17729	:	NCErrorSTRING :='"Axis address" Controller does not know its axis, or the axis address has not been initialized.	.';
17730	:	NCErrorSTRING :='"Drive address" Controller does not know its drive, or the drive address has not been initialized.	.';
17744	:	NCErrorSTRING :='"Following error monitoring (position)" With active following error monitoring (position) a following error exceedance has occurred, whose magnitude is greater than the following error window, and whose duration is longer than the parameterized following error filter time.	.';
17745	:	NCErrorSTRING :='"Following error monitoring (velocity)" With active following error monitoring (velocity) a velocity following error exceedance has occurred, whose magnitude is greater than the following error window, and whose duration is longer than the parameterized following error filter time.	.';
17824	:	NCErrorSTRING :='"CONTROLERR_RANGE_AREA_ASIDE"	.';
17825	:	NCErrorSTRING :='"CONTROLERR_RANGE_AREA_BSIDE"	.';
17826	:	NCErrorSTRING :='"CONTROLERR_RANGE_QNENN"	.';
17827	:	NCErrorSTRING :='"CONTROLERR_RANGE_PNENN"	.';
17828	:	NCErrorSTRING :='"CONTROLERR_RANGE_AXISIDPRESP0"	.';
17920	:	NCErrorSTRING :='‘"Drive ID not allowed" The value for the drive ID is not allowed, e.g. because it has already been assigned, is less than or equal to zero, or is greater than 255.	.';
17921	:	NCErrorSTRING :='‘Drive type impermissible’ The value for the drive type is impermissible, since it is not defined.	.';
17922	:	NCErrorSTRING :='‘Drive operating mode impermissible’ The value for the drive operating mode is impermissible (mode 1: standard).	.';
17923	:	NCErrorSTRING :='"Motor polarity inverted?" The flag for the motor polarity is not allowed. Flag 0: Positive motor polarity flag 1: Negative motor polarity	.';
17924	:	NCErrorSTRING :='‘Drift compensation/speed offset (DAC offset)’ The value for the drift compensation (DAC offset) is impermissible.	.';
17925	:	NCErrorSTRING :='‘Reference speed (velocity pre-control)’ The value for the reference speed (also called velocity pilot control) is impermissible.	.';
17926	:	NCErrorSTRING :='‘Reference output in percent’ The value for the reference output in percent is impermissible. The value 1.0 (100 %) usually corresponds to a voltage of 10.0 V.	.';
17927	:	NCErrorSTRING :='‘Quadrant compensation factor’ The value for the quadrant compensation factor is impermissible.	.';
17928	:	NCErrorSTRING :='‘Velocity reference point’ The value for the velocity reference point in percent is impermissible. The value 1.0 corresponds to 100 percent.	.';
17929	:	NCErrorSTRING :='‘Output reference point’ The value for the output reference point in percent is impermissible. The value 1.0 corresponds to 100 percent.	.';
17930	:	NCErrorSTRING :='‘Minimum or maximum output limits (output limitation)’ The value for the minimum and/or maximum output limit is impermissible. This will happen if the range of values is exceeded, the maximum limit is smaller than the minimum limit, or the distance between the minimum and maximum limits is zero.';
17931	:	NCErrorSTRING :='"Parameter “Maximum Value for Output” is Improper The value for the maximum number of output digits of motion controllers (maximum output value) is improper. According to the used interface (e.g. position, velocity or torque/current). Regarding a velocity interface it is often about a signed 16 bit output value (± 32767)."	.';
17932	:	NCErrorSTRING :='"Parameter “Internal Drive Control Word” is Improper The value as Internal Drive Control Word for the NC is improper. In this control word information from the system manager to the NC is contained what is evaluated at the TC start of the NC."	.';
17933	:	NCErrorSTRING :='"Parameter “Internal Timer for RESET Behavior of Motion Controller” is Improper The special parameter that influences the internal timing behavior between the NC motion controller and the IO motion controller is improper."	.';
17934	:	NCErrorSTRING :='"Parameter “Master Motion Controller ID” is Improper The parameter “master motion controller ID” is improper for a further NC motion controller in slave mode.';
17935	:	NCErrorSTRING :='‘Drive torque output scaling impermissible’ The value is impermissible as drive torque output scaling (rotary motor) or as force output scaling (linear motor).	.';
17936	:	NCErrorSTRING :='„Drive velocity output scaling is not allowed“ The value for the drive velocity output scaling is not allowed.	.';
17937	:	NCErrorSTRING :='‘Profi Drive DSC proportional gain Kpc (controller) impermissible’ Positions The value for the Profi Drive DSC position control gain (Kpc factor) is impermissible.	.';
17938	:	NCErrorSTRING :='‘Table ID is impermissible’ The value for the table ID is impermissible.	.';
17939	:	NCErrorSTRING :='‘Table interpolation type is impermissible’ The value is impermissible as the table interpolation type.	.';
17940	:	NCErrorSTRING :='‘Output offset in percent is impermissible’ The value is impermissible as an output offset in percent (+/- 1.0).	.';
17941	:	NCErrorSTRING :='"‘Profi Drive DSC scaling for calculation of “Xerr” (controller) impermissible’ Positions: the value is impermissible as Profi Drive DSC scaling for the calculation of ‘Xerr’."	.';
17942	:	NCErrorSTRING :='‘Drive acceleration output scaling impermissible’ The value is impermissible as drive acceleration/deceleration output scaling.	.';
17943	:	NCErrorSTRING :='‘Drive position output scaling impermissible’ The value is impermissible as drive position output scaling.	.';
17944	:	NCErrorSTRING :='"Parameter “Dead Time Compensation Mode” (Motion Controller) is Invalid The parameter for the mode of dead time compensation of NC motion controllers is invalid (OFF, ON with velocity, ON with velocity and acceleration)."	.';
17945	:	NCErrorSTRING :='"Parameter “Control Bits of Dead Time Compensation” (Motion Controller) is Invalid The parameter for “control bits of dead time compensation” of NC motion controllers is invalid (e.g. relative or absolute time interpretation)."	.';
17946	:	NCErrorSTRING :='"Parameter “Time Shift of Dead Time Compensation” (Motion Controller) is Invalid The parameter for the time shift of dead time compensation (time shift in nanoseconds) of the NC motion controller is invalid."	.';
17947	:	NCErrorSTRING :='"Parameter “Output Delay (Velocity)” is Invalid The parameter for an optional output delay within the velocity interface to the motion controller is invalid (output delay (velocity)). The maximum permitted delay time has to be smaller than 100 times the NC SAF cycle time."	.';
17948	:	NCErrorSTRING :='‘Drive filter type impermissible for command variable filter for the output position’ The value is impermissible as a drive filter type for the smoothing of the output position (command variable filter for the setpoint position).	.';
17949	:	NCErrorSTRING :='‘Drive filter time impermissible for command variable filter for the output position’ The value is impermissible as a drive filter time for the smoothing of the output position (command variable filter for the setpoint position).	.';
17950	:	NCErrorSTRING :='‘Drive filter order impermissible for command variable filter for the output position’ The value is impermissible as a drive filter order (P-Tn) for the smoothing of the output position (command variable filter for the setpoint position).	.';
17952	:	NCErrorSTRING :='‘Bit mask for stepper motor cycle impermissible’ A value of the different stepper motor masks is impermissible for the respective cycle.	.';
17953	:	NCErrorSTRING :='‘Bit mask for stepper motor holding current impermissible’ The value for the stepper motor holding mask is impermissible.	.';
17954	:	NCErrorSTRING :='‘Scaling factor for actual torque (actual current) impermissible’ The value is impermissible as a scaling factor for the actual torque (or actual current).	.';
17955	:	NCErrorSTRING :='‘Filter time for actual torque is impermissible’ The value is impermissible as a filter time for the actual torque (or the actual current) (P-T1 filter).	.';
17956	:	NCErrorSTRING :='‘Filter time for the temporal derivation of the actual torque is impermissible’ The value is impermissible as a filter time for the temporal derivation of the actual torque (or actual current (P-T1 filter).	.';
17957	:	NCErrorSTRING :='"Parameter for the “Motion Controller Operation Mode” is Invalid The parameter for the motion controller operation mode (position mode, velocity mode, torque mode, …) is invalid.';
17958	:	NCErrorSTRING :='"Motion Controller Functionality is Not Supported A motion controller functionality has been set off that has not been released for usage or has not been implemented (e.g. writing or reading of a motion controller mode that is not supported by certain motion controllers).';
17959	:	NCErrorSTRING :='DRIVEOPERATIONMODEBUSY. The activation of the motion controller controlling mode has failed because another object with OID… uses this interface already.	.';
17960	:	NCErrorSTRING :='"Motion Controller Operation Mode Switching has not been configured or the desired motion controller operation mode cannot be found There has not any motion controller operation mode switching been configured and thus no reading or writing of a motion controller operation mode is possible.';
17968	:	NCErrorSTRING :='‘Overtemperature’ Overtemperature was detected or reported in the drive or terminal.	.';
17969	:	NCErrorSTRING :='‘Undervoltage’ Undervoltage was detected or reported in the drive or terminal.	.';
17970	:	NCErrorSTRING :='‘Wire break in phase A’ A wire break in phase A was detected or reported in the drive or terminal.	.';
17971	:	NCErrorSTRING :='‘Wire break in phase B’ A wire break in phase B was detected or reported in the drive or terminal.	.';
17972	:	NCErrorSTRING :='‘Overcurrent in phase A’ Overcurrent was detected or reported in phase A in the drive or terminal.	.';
17973	:	NCErrorSTRING :='‘Overcurrent in phase B’ Overcurrent was detected or reported in phase B in the drive or terminal.	.';
17974	:	NCErrorSTRING :='‘Torque overload (stall)’ A torque overload (stall) was detected or reported in the drive or terminal.	.';
17984	:	NCErrorSTRING :='‘Drive initialization’ Drive has not been initialized.  Although the drive has been created, the rest of the initialization has not been performed (1. Initialization of drive I/O, 2. Initialization of drive, 3. Reset drive).	.';
17985	:	NCErrorSTRING :='‘Axis address’ Drive does not know its axis, or the axis address has not been initialized.	.';
17986	:	NCErrorSTRING :='‘Address IO input structure’ Drive has no valid IO input address in the process image.	.';
17987	:	NCErrorSTRING :='‘Address IO output structure’ Drive has no valid IO output address in the process image.	.';
18000	:	NCErrorSTRING :='Drive hardware not ready to operate - the drive is in the error state (hardware error)';
18001	:	NCErrorSTRING :='Error in the cyclic communication OF the drive (Life Counter). Reasons FOR THIS could be an interrupted fieldbus OR a drive that is in the error state.	.';
18002	:	NCErrorSTRING :='‘Changing the table ID when active controller enable is impermissible’. Changing (deselecting, selecting) the characteristic curve table ID is not permissible when the controller enable for the axis is active.	.';
18005	:	NCErrorSTRING :='"‘Invalid IO data for more than ‘n’ continuous NC cycles’ The axis (encoder or drive) has detected invalid IO data (e.g. n=3) for more than ‘n’ continuous NC cycles (NC SAF task).';
18944	:	NCErrorSTRING :='"Table ID not allowed" The value for the table ID is not allowed, e.g. because it has already been assigned, is less than or equal to zero, or is greater than 255.	.';
18945	:	NCErrorSTRING :='"Table type not allowed" The value for the table type is unacceptable because it is not defined.	.';
18946	:	NCErrorSTRING :='"Number of lines in the table not allowed" The value of the number of lines in the table is not allowed, because, for example, it is smaller than two at linear interpolation and smaller than four at spline interpolation.	.';
18947	:	NCErrorSTRING :='"Number of columns in the table is not allowed" The value of the number of columns in the table is not allowed, because, for example, it is less than or equal to zero (depends upon the type of table or slave).	.';
18948	:	NCErrorSTRING :='"Step size (position delta) not allowed" The value for the step size between two lines (position delta) is not allowed, because, for example, it is less than or equal to zero.	.';
18949	:	NCErrorSTRING :='"Period not allowed" The value for the period is not allowed, because, for example, it is less than or equal to zero.	.';
18950	:	NCErrorSTRING :='"Table is not monotonic" The value for the step size is not allowed, because, for example, it is less than or equal to zero.	.';
18951	:	NCErrorSTRING :='„Table sub type is not allowed“ The value for the table sub type is not allowed or otherwise the table class (slave type) do not match up to the table main type. Table sub type: (1) equidistant linear position table, (2) equidistant cyclic position table, (3) none equidistant linear position table, (4) none equidistant cyclic position table	.';
18952	:	NCErrorSTRING :='„Table interpolation type is not allowed“ The value for the table interpolation type is allowed. Table interpolation type: (0) linear-interpolation, (1) 4-point-interpolation, (2) spline-interpolation	.';
18953	:	NCErrorSTRING :='"Incorrect table main type" The table main type is unknown or otherwise the table class (slave type) do not match up to the table main type. Table main type: (1) camming table, (2) characteristic table, (3) motion function table (MF)	.';
18960	:	NCErrorSTRING :='"Table initialization" Table has not been initialized. Although the table has been created, the rest of the initialization has not been performed. For instance, the number of lines or columns may be less than or equal to zero.	.';
18961	:	NCErrorSTRING :='"Not enough memory" Table could not be created, since there is not enough memory.	.';
18962	:	NCErrorSTRING :='"Function not executed, function not available" The function has not been implemented, or cannot be executed, for the present type of table.	.';
18963	:	NCErrorSTRING :='"Line index not allowed" The start line index or the stop line index to be used for read or write access to the table is not allowed. For instance, the line index may be greater than the total number of lines in the table.	.';
18964	:	NCErrorSTRING :='"Column index not allowed" The start column index or the stop column index to be used for read or write access to the table in not allowed. For instance, the column index may be greater than the total number of columns in the table.	.';
18965	:	NCErrorSTRING :='"Number of lines not allowed" The number of lines to be read from or written to the table is not allowed. The number of lines must be an integer multiple of the number of elements in a line (n * number of columns).	.';
18966	:	NCErrorSTRING :='"Number of columns not allowed" The number of columns to be read from or written to the table is not allowed. The number of columns must be an integer multiple of the number of elements in a column (n * number of lines).	.';
18967	:	NCErrorSTRING :='"Error in scaling or in range entry" The entries in the table header are inconsistent, e.g. the validity range is empty. If the error is generated during the run time it is a run time error and stops the master/slave group.	.';
18968	:	NCErrorSTRING :='"Multi table slave out of range" The slave master position is outside the table values for the master. The error is a run- time error, and stops the master/slave group.	.';
18969	:	NCErrorSTRING :='"Solo table underflow" The slave master position is outside the table values for the master. The master value of the equidistant table, to be processed linearly, lies under the first table value. The error is a run-time error, and stops the master/slave group.	.';
18970	:	NCErrorSTRING :='"Solo table overflow" The slave master position is outside the table values for the master. The master value of the equidistant table, to be processed linearly, lies above the first table value. The error is a run-time error, and stops the master/slave group.	.';
18971	:	NCErrorSTRING :='"Incorrect execution mode" The cyclic execution mode can only be "true" or "false".	.';
18972	:	NCErrorSTRING :='"Impermissible parameter" The Fifo parameter is not allowed.	.';
18973	:	NCErrorSTRING :='"Fifo is empty" The Fifo of the external generator is empty. This can signify end of track or a run time error.	.';
18974	:	NCErrorSTRING :='"Fifo is full" The Fifo of the external generator is full. It is the user‘s task to continue to attempt to fill the Fifo with the rejected values.	.';
18975	:	NCErrorSTRING :='"„Point-Index of Motion Function invalid“ The point index of a Motion Function Point of a Function Table is invalid. First the point index has to be larger than zero and second it has to be numerical continuously for one column in the Motion Function Table';
18976	:	NCErrorSTRING :='„No diagonalization of matrix“ The spline can not be calculated. The master positions are not correct.	.';
18977	:	NCErrorSTRING :='„Number of spline points to less“ The number of points of a cubic spline has to be greater than two.	.';
18978	:	NCErrorSTRING :='„Fifo must not be overwritten“ Fifo must not be overwritten since then the active line would be overwritten. It is the task of the user to secure that the active line is not modified.	.';
18979	:	NCErrorSTRING :='„Insufficient number of Motion Function points“ The number of valid Motion Function points is less than two. Either the entire number of points is to low or the point type of many points is set to Ignore Point.	.';
19200	:	NCErrorSTRING :='"Axis was stopped" The axis was stopped during travel to the target position. The axis may have been stopped with a PLC command via ADS, a call via AXFNC, or by the System Manager.	.';
19201	:	NCErrorSTRING :='"Axis cannot be started"';
19202	:	NCErrorSTRING :='"Control mode not permitted" No target position control, and no position range control.	.';
19203	:	NCErrorSTRING :='"Axis is not moving" The position and velocity can only be restarted while the axis is physically in motion.	.';
19204	:	NCErrorSTRING :='"“Invalid Mode” Examples: Invalid Direction input to MC_MoveModulo. Inactive axis parameter position correction for MC_BacklashCompensation."	.';
19205	:	NCErrorSTRING :='"Command not permitted"" •  Continuous motion in an unspecified direction •  Read/Write parameters: type mismatch"	.';
19206	:	NCErrorSTRING :='"Parameter incorrect"" •  Incorrect override: > 100% or < 0% •  Incorrect gear ratio: RatioDenominator = 0".';
19207	:	NCErrorSTRING :='"Timeout axis function block"" After positioning, all ""MC_Move..."" blocks check whether positioning was completed successfully. In the simplest case, the ""AxisHasJob"" flag of the NC axis is checked, which initially signifies that positioning was logically completed. ';
19208	:	NCErrorSTRING :='"Axis is in protected mode" The axis is in protected mode ( e.g. coupled) and cannot be moved.	.';
19209	:	NCErrorSTRING :='"Axis is not ready" The axis is not ready and cannot be moved.	.';
19210	:	NCErrorSTRING :='"Error during referencing" Referencing (homing) of the axis could not be started or was not successful.	.';
19211	:	NCErrorSTRING :='"Incorrect definition of the trigger input" The definition of the trigger signal for block MC_TouchProbe is incorrect. The defined encoder-ID, the trigger signal or the trigger edge are invalid.	.';
19212	:	NCErrorSTRING :='"Position latch was disabled" The function block MC_TouchProbe has detected that a measuring probe cycle it had started was disabled. The reason may be an axis reset, for example.	.';
19213	:	NCErrorSTRING :='‘NC status feedback timeout’  A function was successfully sent from the PLC to the NC. An expected feedback in the axis status word has not arrived.	.';
19214	:	NCErrorSTRING :='"Additional product not installed" The function is available as an additional product but is not installed on the system.	.';
19215	:	NCErrorSTRING :='"No NC Cycle Counter Update" – The NcToPlc Interface or the NC Cycle Counter in the NcToPlc Interface was not updated.	.';
19216	:	NCErrorSTRING :='"M-function query missing" This error occurs if the M- function was confirmed, but the request bit was not set.	.';
19217	:	NCErrorSTRING :='"Zero offset index is outside the range" The index of the zero offset is invalid.	.';
19218	:	NCErrorSTRING :='"R-parameter index or size is invalid" This error occurs if the R-parameters are written or read but the index or size are outside the range.	.';
19219	:	NCErrorSTRING :='"Index for tool description is invalid"	.';
19220	:	NCErrorSTRING :='"Version of the cyclic channel interface does not match the requested function or the function block" This error occurs if an older TwinCAT version is used to call new functions of a later TcNci.lib version.	.';
19221	:	NCErrorSTRING :='"Channel is not ready for the requested function" The requested function cannot be executed, because the channel is in the wrong state. This error occurs during reverse travel, for example, if the axis was not stopped with ItpEStop first.	.';
19222	:	NCErrorSTRING :='"Requested function is not activated" The requested function requires explicit activation.	.';
19223	:	NCErrorSTRING :='"Axis is already in another group" The axis has already been added to another group.	.';
19224	:	NCErrorSTRING :='"Block search could not be executed successfully"" The block search has failed. ';
19225	:	NCErrorSTRING :='"Invalid block search parameter" This error occurs if the FB ItpBlocksearch is called with invalid parameters (e.g. E_ItpDryRunMode, E_ItpBlockSearchMode)	.';
19232	:	NCErrorSTRING :='"Cannot add all axes" This error occurs if an auxiliary axis is to be added to an interpolation group, but the function fails. It is likely that a preceding instruction of an auxiliary axis was skipped.	.';
19248	:	NCErrorSTRING :='"Pointer is invalid"" A pointer to a data structure is invalid, e.g. Null•  Data structure MC_CAM_REF was not initialized"	.';
19249	:	NCErrorSTRING :='"Memory size invalid"" The specification of the memory size (SIZE) for a data structure is invalid.';
19250	:	NCErrorSTRING :='"Cam table ID is invalid" The ID of a cam table is not between 1 and 255.	.';
19251	:	NCErrorSTRING :='"Point ID is invalid" The ID of a point (sampling point) of a motion function is less than 1.	.';
19252	:	NCErrorSTRING :='"Number of points is invalid" The number of points (sampling points) of a cam plate to be read or written is less than 1.	.';
19253	:	NCErrorSTRING :='"MC table type is invalid" The type of a cam plate does not match the definition MC_TableType.	.';
19254	:	NCErrorSTRING :='"Number of rows invalid" The number of rows (sampling points) of a cam table is less than 1.	.';
19255	:	NCErrorSTRING :='"Number of columns invalid"" The number of columns of a cam table is invalid.';
19256	:	NCErrorSTRING :='"Step size invalid". The increment for the interpolation is invalid, e.g. less than or equal to zero.	.';
19264	:	NCErrorSTRING :='"Terminal type not supported" The terminal used is not supported by this function block.	.';
19265	:	NCErrorSTRING :='"Register read/write error" This error implies a validity error.	.';
19266	:	NCErrorSTRING :='"Axis is enabled" The axis is enabled but should not be enabled for this process.	.';
19267	:	NCErrorSTRING :='"Incorrect size of the compensation table" The specified table size (in bytes) does not match the actual size	.';
19268	:	NCErrorSTRING :='The minimum/maximum position in the compensation table does not match the position in the table description (ST_CompensationDesc)	.';
19269	:	NCErrorSTRING :='"Not implemented" The requested function is not implemented in this combination	.';
19296	:	NCErrorSTRING :='"Motion command did not become active" A motion command has been started and has been buffered and confirmed by the NC. Nevertheless, the motion command did not become active (possibly due to a terminating condition or an internal NC error).	.';
19297	:	NCErrorSTRING :='"Motion command could not be monitored by the PLC" A motion command has been started and has been buffered and confirmed by the NC. The PLC has not been able to monitor the execution of this command and the execution status is unclear since the NC is already executing a more recent command.';
19298	:	NCErrorSTRING :='"Buffered command was terminated with an error" A buffered command was terminated with an error. The error number is not available, because a new command is already being executed.	.';
19299	:	NCErrorSTRING :='"Buffered command was completed without feedback" A buffered command was completed but there was no feedback to indicate success or failure.	.';
19300	:	NCErrorSTRING :='"BufferMode is not supported by the command" The BufferMode is not supported by this command.	.';
19301	:	NCErrorSTRING :='"Command number is zero" The command number for queued commands managed by the system unexpectedly has the value 0.	.';
19302	:	NCErrorSTRING :='"Function block was not called cyclically" The function block was not called cyclically. The command execution could not be monitored by the PLC, because the NC was already executing a subsequent command. The execution state is unclear.	.';
19313	:	NCErrorSTRING :='"Invalid NCI entry type". The FB FB_NciFeedTablePreparation was called with an unknown nEntryType.	.';
19314	:	NCErrorSTRING :='"NCI feed table full"" The table is full, and the entry is therefore not accepted.';
19315	:	NCErrorSTRING :='INTERNAL error	.';
19316	:	NCErrorSTRING :='"ST_NciTangentialFollowingDesc: tangential axis is not an auxiliary axis" The entry for tangential following contains a tangential axis that is not an auxiliary axis.	.';
19317	:	NCErrorSTRING :='ST_NciTangentialFollowingDesc: nPathAxis1 or nPathAxis2 is not a path axis. It is therefore not possible to determine the plane.	.';
19318	:	NCErrorSTRING :='ST_NciTangentialFollwoingDesc: nPathAxis1 and nPathAxis2 are the same. It is therefore not possible to determine the plane.	.';
19319	:	NCErrorSTRING :='ST_NciGeoCirclePlane: Circle incorrectly parameterized	.';
19320	:	NCErrorSTRING :='Internal error during calculation of tangential following	.';
19321	:	NCErrorSTRING :='Tangential following: Monitoring of the deviation angle was activated during activation of tangential following (E_TfErrorOnCritical1), and an excessively large deviation angle was detected in the current segment.	.';
19322	:	NCErrorSTRING :='not implemented	.';
19323	:	NCErrorSTRING :='Tangential following: the radius of the current arc is too small	.';
19324	:	NCErrorSTRING :='FB_NciFeedTablePreparation: pEntry is NULL	.';
19325	:	NCErrorSTRING :='FB_NciFeedTablePreparation: the specified nEntryType does not match the structure type	.';
19326	:	NCErrorSTRING :='ST_NciMFuncFast and ST_NciMFuncHsk: the requested M-function is not between 0 and 159	.';
19327	:	NCErrorSTRING :='ST_NciDynOvr: the requested value for the dynamic override is not between 0.01 and 1	.';
19328	:	NCErrorSTRING :='ST_NciVertexSmoothing: invalid parameter. This error is generated if a negative smoothing radius or an unknown smoothing type is encountered.	.';
19329	:	NCErrorSTRING :='FB_NciFeedTablePrepartion: The requested velocity is not in the valid range	.';
19330	:	NCErrorSTRING :='ST_Nci*: invalid parameter	.';
19344	:	NCErrorSTRING :='Determined drive type is not supported	.';
19345	:	NCErrorSTRING :='Direction is impermissible	.';
19346	:	NCErrorSTRING :='SwitchMode is impermissible	.';
19347	:	NCErrorSTRING :='Mode for the parameter handling is impermissible	.';
19348	:	NCErrorSTRING :='Parameterization of the torque limits is inconsistent	.';
19349	:	NCErrorSTRING :='Parameterization of the position lag limit is impermissible (<=0).	.';
19350	:	NCErrorSTRING :='Parameterization of the distance limit is impermissible (<0)	.';
19351	:	NCErrorSTRING :='An attempt was made to back up parameters again, although they have already been backed up.	.';
19352	:	NCErrorSTRING :='An attempt was made to restore parameters, although none have been backed up.	.';
19360	:	NCErrorSTRING :='"KinGroup error: the kinematic group is in an error state. This error may occur if the kinematic group is in an error state or an unexpected state when it is called (e.g. simultaneous call via several FB instances)."	.';
19361	:	NCErrorSTRING :='KinGroup timeout: timeout during call of a kinematic block	.';
19376	:	NCErrorSTRING :='The current axis position or the axis position resulting from the new position offset exceeds the valid range of values.	.';
19377	:	NCErrorSTRING :='The new position offset exceeds the valid range of values [AX5000: 2^31]	.';
19378	:	NCErrorSTRING :='The current axis position or the axis position resulting from the new position offset falls below the valid range of values.	.';
19379	:	NCErrorSTRING :='The new position offset falls below the valid range of values [AX5000: -2^31]	.';
19380	:	NCErrorSTRING :='The activated feedback and/or storage location (AX5000: P-0-0275) differ from the parameterization on the function block.	.';
19381	:	NCErrorSTRING :='"Reinitialisation of the Nc actual position has failed. e.g. reference system = “ABSOLUTE (with single overflow)” & software end position monitoring is disabled."	.';
19382	:	NCErrorSTRING :='"The command for setting or deleting a position offset has been rejected without sending feedback data. E.g. if the motion controller firmware does not support the corresponding command."	.';
19383	:	NCErrorSTRING :='"The command for setting or deleting a position offset has been rejected with sending feedback data. Informations within the feedback data may contain further indications on the origin of the error. E.g. if the motion controller firmware does not support the corresponding command';
19456	:	NCErrorSTRING :='Transformation failed.	.';
19457	:	NCErrorSTRING :='Ambiguous answer. The answer of the transformation is not explicit.	.';
19458	:	NCErrorSTRING :='"Invalid axis position: The transformation can not be calculated with the current position data.';
19459	:	NCErrorSTRING :='"Invalid dimension: The dimension of the paramerterized input parameter does not match the dimension expected by the kinematic object.';
19460	:	NCErrorSTRING :='NCERR_KINTRAFO_REGISTRATION	.';
19461	:	NCErrorSTRING :='Newton iteration failed: The Newton iteration does not converge.	.';
19462	:	NCErrorSTRING :='Jacobi matrix cannot be inverted	.';
19463	:	NCErrorSTRING :='Invalid cascade: This kinematic configuration is not permitted.	.';
19464	:	NCErrorSTRING :='Singularity: The machine configuration results in singular axis velocities.	.';
19467	:	NCErrorSTRING :='No metainfo: Metainfo pointer is null.	.';
19475	:	NCErrorSTRING :='"NCERR_RBTFRAME_INVALIDWCSTOMCS, The employed WcsToMcs component leads to positions that the selected kinematics cannot adopt to. Tailoring the WcsToMcs parameters is required."	.';
19488	:	NCErrorSTRING :='Transformation failed: Call of extended kinematic model failed.	.';
19504	:	NCErrorSTRING :='Invalid input frame: Programmed Cartesian position cannot be reached in the ACS configuration.	.';
19536	:	NCErrorSTRING :='Invalid Offset: Access violation within the observer detected.	.';
ELSE
	NCErrorSTRING :='Error not defined';
END_CASE
FUN_NC_FindErrorText := NCErrorSTRING;

END_FUNCTION

(* stored: Version 1.1.0.1, ProductVersion 3.1.4024.14
   POU FUN_NC_FindErrorText: Id {0e7ee97e-2696-49d0-8819-1ff85bc49730}, SpecialFunc None *)
